// TwinCAT 3 PLC project Linearachse
// ProgramVersion: 3.1.4022.1
// libraries:
//   Tc2_Standard, * (Beckhoff Automation GmbH)
//   Tc2_System, * (Beckhoff Automation GmbH)
//   Tc3_Module, * (Beckhoff Automation GmbH)
// project tree:
//   GVLs/ dSub.TcGVL
//   / PlcTask.TcTTO (not stored)
//   POUs/ Linearachse.TcPOU (not stored), MAIN.TcPOU (not stored)

// ---- GVLs/dSub.TcGVL
{attribute 'qualified_only'}
VAR_GLOBAL
	
	// Linearantrieb Endlage links (Öffner)
	B1 AT %I*: BOOL; 
	// Linearantrieb Endlage rechts (Öffner)
	B2 AT %I*: BOOL;
	// Taster (1) (Schliesser)
	S1 AT %I*: BOOL;		
	// Taster (0) (Öffner)
	S2 AT %I*: BOOL;
	// Taster I (Schliesser)
	S3 AT %I*: BOOL;
	// Taster II (Schliesser)
	S4 AT %I*: BOOL;
	// Taster Pfeil auf (Schliesser)
	S5 AT %I*: BOOL;
	// Taster Pfeil ab (Schliesser)
	S6 AT %I*: BOOL;
	// Taster + (Schliesser)
	S7 AT %I*: BOOL;
	// Taster - (Schliesser)
	S8 AT %I*: BOOL;
	// Taster STOP (Öffner)
	S9 AT %I*: BOOL;
	// Taster Not Halt (Öffner)
	S10 AT %I*: BOOL;
	// Taster Not Halt (Schliesser)
	S11 AT %I*: BOOL;

	// Linearantrieb Rechtslauf
	Q1 AT %Q*: BOOL;
	// Linearantrieb Linkslauf
	Q2 AT %Q*: BOOL;
	// Meldeleuchte im Taster S1 (weiß)
	P1 AT %Q*: BOOL;
	// Meldeleuchte weiß
	P2 AT %Q*: BOOL;
	// Meldeleuchte rot
	P3 AT %Q*: BOOL;
	// Meldeleuchte grün
	P4 AT %Q*: BOOL;

END_VAR
